SUBAPPLICATION Uebung_003c (* DigitalInput_I1-2-3-4 auf AUX *)
  (* Standard: 61499-2; Description: Copyright (c) 2023 Meisterschulen am Ostbahnhof This program and the accompanying materials are made available under the terms of the Eclipse Public License 2.0 which is available at https://www.eclipse.org/legal/epl-2.0/ SPDX-License-Identifier: EPL-2.0 *)
  (* Version 1.0, 2023-10-23, Franz Höpfinger, Meisterschulen am Ostbahnhof *)
  PACKAGE Uebungen;
  IMPORT logiBUS::io::DI::logiBUS_DI::Input_I1;
  IMPORT logiBUS::io::DI::logiBUS_DI::Input_I2;
  IMPORT logiBUS::io::DI::logiBUS_DI::Input_I3;
  IMPORT logiBUS::io::DI::logiBUS_DI::Input_I4;
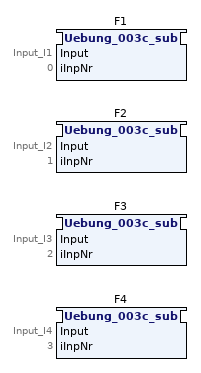
  SUBAPPS
    F1 : Uebungen::Uebung_003c_sub(Input := Input_I1, iInpNr := 0);
    F2 : Uebungen::Uebung_003c_sub(Input := Input_I2, iInpNr := 1);
    F3 : Uebungen::Uebung_003c_sub(Input := Input_I3, iInpNr := 2);
    F4 : Uebungen::Uebung_003c_sub(Input := Input_I4, iInpNr := 3);
  END_SUBAPPS
END_SUBAPPLICATION
